// TIA Portal V19 export
FUNCTION "OUTPUT MAPING" : Void   // FC2, LAD
{ S7_Optimized_Access := 'TRUE' }
// stored: SetENOAutomatically false
BEGIN

REGION Network 1: "P-202 A RO 1 FEED PUMP"
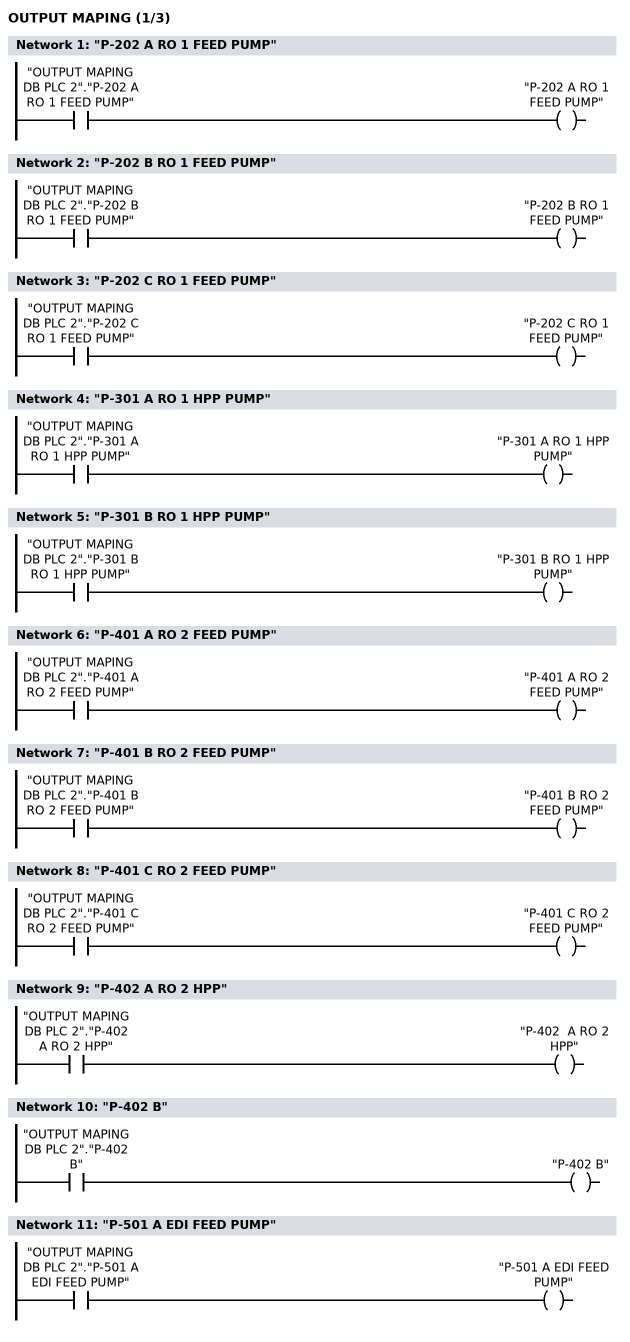
   RUNG wire#powerrail
      Contact( "OUTPUT MAPING DB PLC 2"."P-202 A RO 1 FEED PUMP" )
      Coil( "P-202 A RO 1 FEED PUMP" )
   END_RUNG
   // the same network as SCL:
   "P-202 A RO 1 FEED PUMP" := "OUTPUT MAPING DB PLC 2"."P-202 A RO 1 FEED PUMP";
END_REGION

REGION Network 2: "P-202 B RO 1 FEED PUMP"
   RUNG wire#powerrail
      Contact( "OUTPUT MAPING DB PLC 2"."P-202 B RO 1 FEED PUMP" )
      Coil( "P-202 B RO 1 FEED PUMP" )
   END_RUNG
   // the same network as SCL:
   "P-202 B RO 1 FEED PUMP" := "OUTPUT MAPING DB PLC 2"."P-202 B RO 1 FEED PUMP";
END_REGION

REGION Network 3: "P-202 C RO 1 FEED PUMP"
   RUNG wire#powerrail
      Contact( "OUTPUT MAPING DB PLC 2"."P-202 C RO 1 FEED PUMP" )
      Coil( "P-202 C RO 1 FEED PUMP" )
   END_RUNG
   // the same network as SCL:
   "P-202 C RO 1 FEED PUMP" := "OUTPUT MAPING DB PLC 2"."P-202 C RO 1 FEED PUMP";
END_REGION

REGION Network 4: "P-301 A RO 1 HPP PUMP"
   RUNG wire#powerrail
      Contact( "OUTPUT MAPING DB PLC 2"."P-301 A RO 1 HPP PUMP" )
      Coil( "P-301 A RO 1 HPP PUMP" )
   END_RUNG
   // the same network as SCL:
   "P-301 A RO 1 HPP PUMP" := "OUTPUT MAPING DB PLC 2"."P-301 A RO 1 HPP PUMP";
END_REGION

REGION Network 5: "P-301 B RO 1 HPP PUMP"
   RUNG wire#powerrail
      Contact( "OUTPUT MAPING DB PLC 2"."P-301 B RO 1 HPP PUMP" )
      Coil( "P-301 B RO 1 HPP PUMP" )
   END_RUNG
   // the same network as SCL:
   "P-301 B RO 1 HPP PUMP" := "OUTPUT MAPING DB PLC 2"."P-301 B RO 1 HPP PUMP";
END_REGION

REGION Network 6: "P-401 A RO 2 FEED PUMP"
   RUNG wire#powerrail
      Contact( "OUTPUT MAPING DB PLC 2"."P-401 A RO 2 FEED PUMP" )
      Coil( "P-401 A RO 2 FEED PUMP" )
   END_RUNG
   // the same network as SCL:
   "P-401 A RO 2 FEED PUMP" := "OUTPUT MAPING DB PLC 2"."P-401 A RO 2 FEED PUMP";
END_REGION

REGION Network 7: "P-401 B RO 2 FEED PUMP"
   RUNG wire#powerrail
      Contact( "OUTPUT MAPING DB PLC 2"."P-401 B RO 2 FEED PUMP" )
      Coil( "P-401 B RO 2 FEED PUMP" )
   END_RUNG
   // the same network as SCL:
   "P-401 B RO 2 FEED PUMP" := "OUTPUT MAPING DB PLC 2"."P-401 B RO 2 FEED PUMP";
END_REGION

REGION Network 8: "P-401 C RO 2 FEED PUMP"
   RUNG wire#powerrail
      Contact( "OUTPUT MAPING DB PLC 2"."P-401 C RO 2 FEED PUMP" )
      Coil( "P-401 C RO 2 FEED PUMP" )
   END_RUNG
   // the same network as SCL:
   "P-401 C RO 2 FEED PUMP" := "OUTPUT MAPING DB PLC 2"."P-401 C RO 2 FEED PUMP";
END_REGION

REGION Network 9: "P-402 A RO 2 HPP"
   RUNG wire#powerrail
      Contact( "OUTPUT MAPING DB PLC 2"."P-402  A RO 2 HPP" )
      Coil( "P-402  A RO 2 HPP" )
   END_RUNG
   // the same network as SCL:
   "P-402  A RO 2 HPP" := "OUTPUT MAPING DB PLC 2"."P-402  A RO 2 HPP";
END_REGION

REGION Network 10: "P-402 B"
   RUNG wire#powerrail
      Contact( "OUTPUT MAPING DB PLC 2"."P-402 B" )
      Coil( "P-402 B" )
   END_RUNG
   // the same network as SCL:
   "P-402 B" := "OUTPUT MAPING DB PLC 2"."P-402 B";
END_REGION

REGION Network 11: "P-501 A EDI FEED PUMP"
   RUNG wire#powerrail
      Contact( "OUTPUT MAPING DB PLC 2"."P-501 A EDI FEED PUMP" )
      Coil( "P-501 A EDI FEED PUMP" )
   END_RUNG
   // the same network as SCL:
   "P-501 A EDI FEED PUMP" := "OUTPUT MAPING DB PLC 2"."P-501 A EDI FEED PUMP";
END_REGION

REGION Network 12: "P-501 B EDI FEED PUMP"
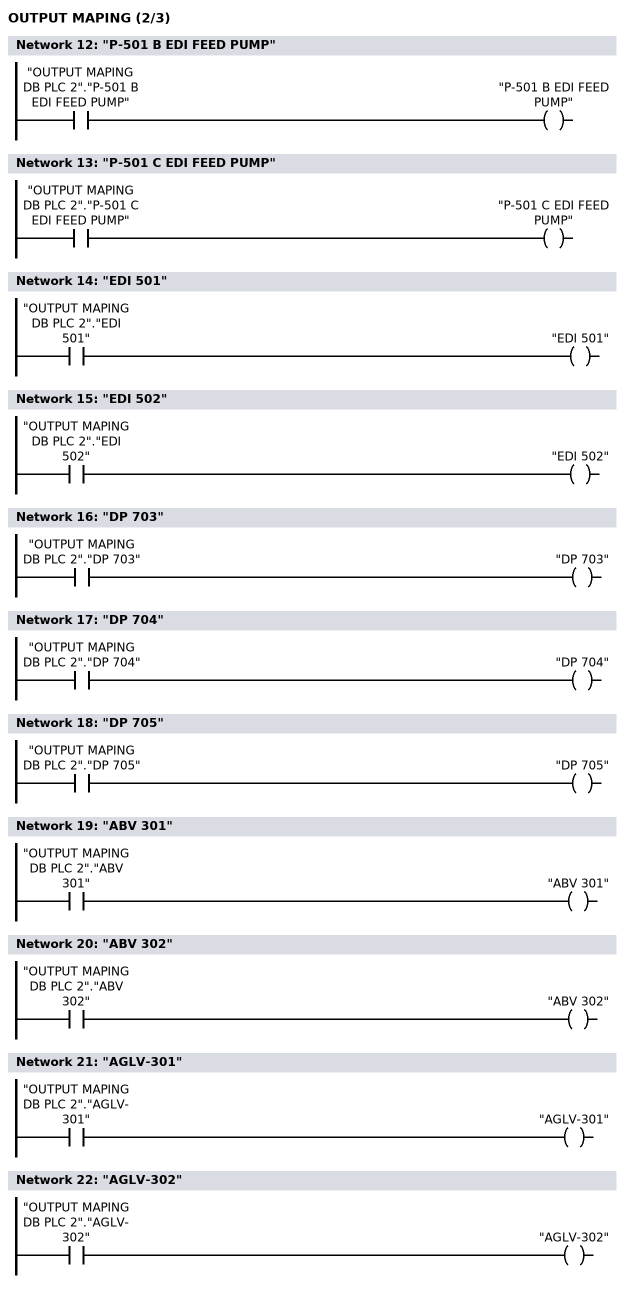
   RUNG wire#powerrail
      Contact( "OUTPUT MAPING DB PLC 2"."P-501 B EDI FEED PUMP" )
      Coil( "P-501 B EDI FEED PUMP" )
   END_RUNG
   // the same network as SCL:
   "P-501 B EDI FEED PUMP" := "OUTPUT MAPING DB PLC 2"."P-501 B EDI FEED PUMP";
END_REGION

REGION Network 13: "P-501 C EDI FEED PUMP"
   RUNG wire#powerrail
      Contact( "OUTPUT MAPING DB PLC 2"."P-501 C EDI FEED PUMP" )
      Coil( "P-501 C EDI FEED PUMP" )
   END_RUNG
   // the same network as SCL:
   "P-501 C EDI FEED PUMP" := "OUTPUT MAPING DB PLC 2"."P-501 C EDI FEED PUMP";
END_REGION

REGION Network 14: "EDI 501"
   RUNG wire#powerrail
      Contact( "OUTPUT MAPING DB PLC 2"."EDI 501" )
      Coil( "EDI 501" )
   END_RUNG
   // the same network as SCL:
   "EDI 501" := "OUTPUT MAPING DB PLC 2"."EDI 501";
END_REGION

REGION Network 15: "EDI 502"
   RUNG wire#powerrail
      Contact( "OUTPUT MAPING DB PLC 2"."EDI 502" )
      Coil( "EDI 502" )
   END_RUNG
   // the same network as SCL:
   "EDI 502" := "OUTPUT MAPING DB PLC 2"."EDI 502";
END_REGION

REGION Network 16: "DP 703"
   RUNG wire#powerrail
      Contact( "OUTPUT MAPING DB PLC 2"."DP 703" )
      Coil( "DP 703" )
   END_RUNG
   // the same network as SCL:
   "DP 703" := "OUTPUT MAPING DB PLC 2"."DP 703";
END_REGION

REGION Network 17: "DP 704"
   RUNG wire#powerrail
      Contact( "OUTPUT MAPING DB PLC 2"."DP 704" )
      Coil( "DP 704" )
   END_RUNG
   // the same network as SCL:
   "DP 704" := "OUTPUT MAPING DB PLC 2"."DP 704";
END_REGION

REGION Network 18: "DP 705"
   RUNG wire#powerrail
      Contact( "OUTPUT MAPING DB PLC 2"."DP 705" )
      Coil( "DP 705" )
   END_RUNG
   // the same network as SCL:
   "DP 705" := "OUTPUT MAPING DB PLC 2"."DP 705";
END_REGION

REGION Network 19: "ABV 301"
   RUNG wire#powerrail
      Contact( "OUTPUT MAPING DB PLC 2"."ABV 301" )
      Coil( "ABV 301" )
   END_RUNG
   // the same network as SCL:
   "ABV 301" := "OUTPUT MAPING DB PLC 2"."ABV 301";
END_REGION

REGION Network 20: "ABV 302"
   RUNG wire#powerrail
      Contact( "OUTPUT MAPING DB PLC 2"."ABV 302" )
      Coil( "ABV 302" )
   END_RUNG
   // the same network as SCL:
   "ABV 302" := "OUTPUT MAPING DB PLC 2"."ABV 302";
END_REGION

REGION Network 21: "AGLV-301"
   RUNG wire#powerrail
      Contact( "OUTPUT MAPING DB PLC 2"."AGLV-301" )
      Coil( "AGLV-301" )
   END_RUNG
   // the same network as SCL:
   "AGLV-301" := "OUTPUT MAPING DB PLC 2"."AGLV-301";
END_REGION

REGION Network 22: "AGLV-302"
   RUNG wire#powerrail
      Contact( "OUTPUT MAPING DB PLC 2"."AGLV-302" )
      Coil( "AGLV-302" )
   END_RUNG
   // the same network as SCL:
   "AGLV-302" := "OUTPUT MAPING DB PLC 2"."AGLV-302";
END_REGION

REGION Network 23: "AGLV-401"
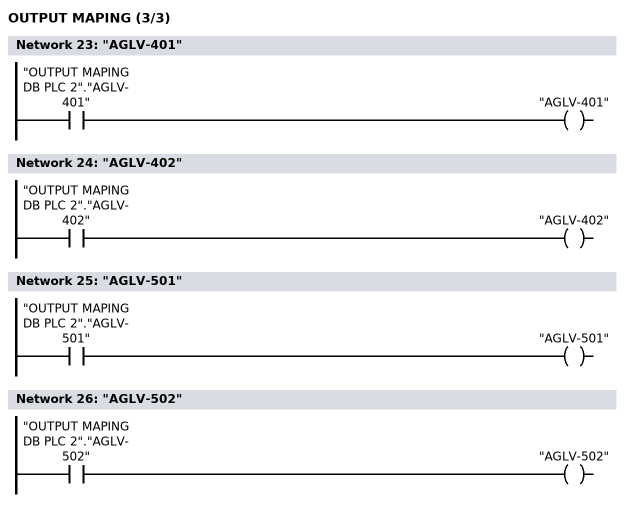
   RUNG wire#powerrail
      Contact( "OUTPUT MAPING DB PLC 2"."AGLV-401" )
      Coil( "AGLV-401" )
   END_RUNG
   // the same network as SCL:
   "AGLV-401" := "OUTPUT MAPING DB PLC 2"."AGLV-401";
END_REGION

REGION Network 24: "AGLV-402"
   RUNG wire#powerrail
      Contact( "OUTPUT MAPING DB PLC 2"."AGLV-402" )
      Coil( "AGLV-402" )
   END_RUNG
   // the same network as SCL:
   "AGLV-402" := "OUTPUT MAPING DB PLC 2"."AGLV-402";
END_REGION

REGION Network 25: "AGLV-501"
   RUNG wire#powerrail
      Contact( "OUTPUT MAPING DB PLC 2"."AGLV-501" )
      Coil( "AGLV-501" )
   END_RUNG
   // the same network as SCL:
   "AGLV-501" := "OUTPUT MAPING DB PLC 2"."AGLV-501";
END_REGION

REGION Network 26: "AGLV-502"
   RUNG wire#powerrail
      Contact( "OUTPUT MAPING DB PLC 2"."AGLV-502" )
      Coil( "AGLV-502" )
   END_RUNG
   // the same network as SCL:
   "AGLV-502" := "OUTPUT MAPING DB PLC 2"."AGLV-502";
END_REGION
END_FUNCTION
